SUBAPPLICATION Uebung_022_AX (* Spiegelabfolge (2) - AX Variante *)
  (* Standard: 61499-2; Description: Copyright (c) 2023 Meisterschulen am Ostbahnhof This program and the accompanying materials are made available under the terms of the Eclipse Public License 2.0 which is available at https://www.eclipse.org/legal/epl-2.0/ SPDX-License-Identifier: EPL-2.0 *)
  (* Version 1.0, 2026-04-20, Franz Höpfinger, Meisterschulen am Ostbahnhof, AX Variante *)
  PACKAGE Uebungen;
  IMPORT Uebungen::const::UT::DefaultPool::SoftKey_F1;
  IMPORT Uebungen::const::UT::DefaultPool::SoftKey_F2;
  IMPORT Uebungen::const::UT::DefaultPool::SoftKey_F3;
  IMPORT logiBUS::io::DQ::logiBUS_DO::Output_Q1;
  IMPORT logiBUS::io::DQ::logiBUS_DO::Output_Q2;
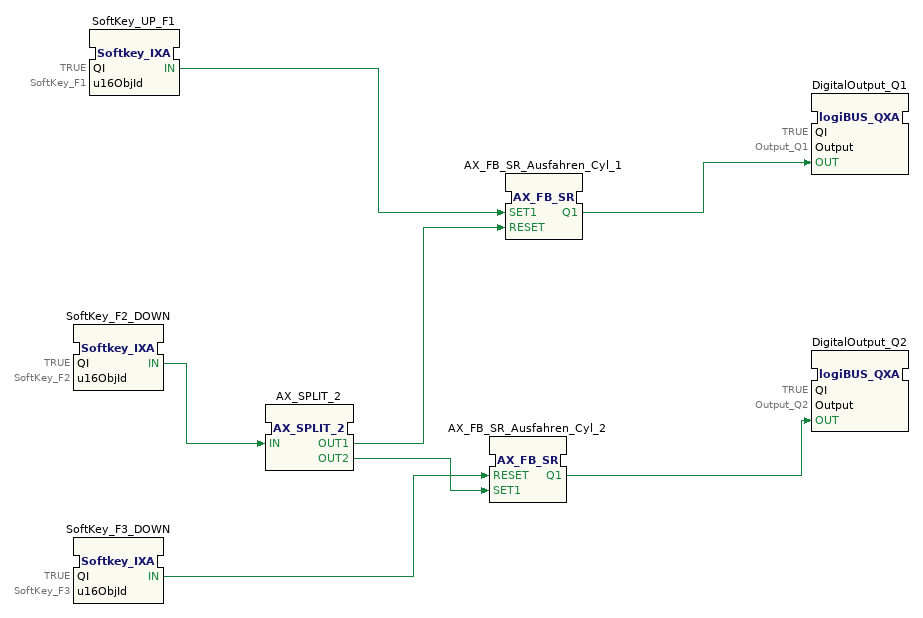
  (* START-Knopf *)
  (* Endlage Ausfahren_Cyl_1 *)
  (* Endlage Ausfahren_Cyl_2 *)
  (* Ausfahren_Cyl_1 *)
  (* Ausfahren_Cyl_2 *)
  FBS
    DigitalOutput_Q1 : logiBUS::io::DQ::logiBUS_QXA(QI := TRUE, Output := Output_Q1);
    SoftKey_UP_F1 : isobus::UT::io::Softkey::Softkey_IXA(QI := TRUE, u16ObjId := SoftKey_F1);
    AX_FB_SR_Ausfahren_Cyl_1 : adapter::iec61131::bistableElements::AX_FB_SR;
    SoftKey_F2_DOWN : isobus::UT::io::Softkey::Softkey_IXA(QI := TRUE, u16ObjId := SoftKey_F2);
    DigitalOutput_Q2 : logiBUS::io::DQ::logiBUS_QXA(QI := TRUE, Output := Output_Q2);
    AX_FB_SR_Ausfahren_Cyl_2 : adapter::iec61131::bistableElements::AX_FB_SR;
    SoftKey_F3_DOWN : isobus::UT::io::Softkey::Softkey_IXA(QI := TRUE, u16ObjId := SoftKey_F3);
    AX_SPLIT_2 : adapter::events::unidirectional::AX_SPLIT_2;
  END_FBS
  ADAPTER_CONNECTIONS
    SoftKey_UP_F1.IN TO AX_FB_SR_Ausfahren_Cyl_1.SET1;
    AX_FB_SR_Ausfahren_Cyl_1.Q1 TO DigitalOutput_Q1.OUT;
    AX_FB_SR_Ausfahren_Cyl_2.Q1 TO DigitalOutput_Q2.OUT;
    SoftKey_F3_DOWN.IN TO AX_FB_SR_Ausfahren_Cyl_2.RESET;
    SoftKey_F2_DOWN.IN TO AX_SPLIT_2.IN;
    AX_SPLIT_2.OUT1 TO AX_FB_SR_Ausfahren_Cyl_1.RESET;
    AX_SPLIT_2.OUT2 TO AX_FB_SR_Ausfahren_Cyl_2.SET1;
  END_CONNECTIONS
END_SUBAPPLICATION
